TYPE Room_Ctx_Io :
STRUCT
	bOpenValves			: BOOL;
	
	bValvesOpen			: BOOL;
	bValvesClosed		: BOOL;
END_STRUCT
END_TYPE

(* stored: Version 1.1.0.1
   DUT Room_Ctx_Io: Id {67371870-bd5d-49c5-aa16-53adf3c88038} *)
